/// Generate time data in different formats.
{attribute: 'hide_all_locals'}
FUNCTION_BLOCK PUBLIC DateTime
VAR
  local_system_time : Tc2_Utilities.FB_LocalSystemTime;
  get_system_time : Tc2_System.GetSystemTime;
  time_zone_info : Tc2_Utilities.FB_GetTimeZoneInformation;
  local_Time : Tc2_Utilities.FB_SystemTimeToTzSpecificLocalTime;
  local_system_time_valid : Tc2_Standard.R_Trig;
  utc_time : Tc2_Utilities.FB_TzSpecificLocalTimeToFileTime;
END_VAR

// Get local system time
local_system_time(
	sNetID  :=  '',
	bEnable :=  TRUE,
	dwCycle :=  1,
	dwOpt :=  1,
	tTimeout:= Tc2_System.Default_Ads_Timeout
);

// Get timezone information
time_zone_info(
	sNetID := '',
	bExecute := TRUE,
	tTimeout := Tc2_System.Default_Ads_Timeout
);

// Convert local time to utc time
utc_time(
	in := THIS^.AsLocalFileTime,
	tzInfo := time_zone_info.tzInfo
);
  
// Finished retrieving time data
local_system_time_valid(Clk := local_system_time.bValid);

/// Returns local time as `Tc2_Utilities.T_FILETIME`.
{attribute 'monitoring':='variable'}
PROPERTY AsLocalFileTime : Tc2_Utilities.T_FILETIME
GET
AsLocalFileTime := SYSTEMTIME_TO_FILETIME(THIS^.AsLocalSystemTime);
END_GET
END_PROPERTY

/// Returns local time as `Tc2_Utilities.TIMESTRUCT`.
{attribute 'monitoring':='variable'}
PROPERTY AsLocalSystemTime : Tc2_Utilities.TIMESTRUCT
GET
AsLocalSystemTime := local_system_time.systemTime;
END_GET
END_PROPERTY

/// Returns local time as string.
{attribute 'monitoring':='variable'}
PROPERTY AsLocalSystemTimeString : Tc2_System.T_MAXSTRING
GET
AsLocalSystemTimeString := Tc2_Utilities.SYSTEMTIME_TO_STRING(THIS^.AsLocalSystemTime);
END_GET
END_PROPERTY

/// Returns UTC time as `Tc2_Utilities.T_FILETIME`.
{attribute 'monitoring':='variable'}
PROPERTY AsUtcFileTime : Tc2_Utilities.T_FILETIME
GET
AsUtcFileTime := utc_time.out;
END_GET
END_PROPERTY

/// When calling `DateTime` the first time, it takes some time until all time and timezone information is available.
/// `Done` is `TRUE` for one cycle, once all the data is ready. 
{attribute 'monitoring':='call'}
PROPERTY Done : BOOL
GET
Done := local_system_time_valid.Q;
END_GET
END_PROPERTY

// Replaces placeholders in format string by the actual time values.
{attribute 'hide_all_locals'}
{attribute 'hide'}
METHOD PRIVATE ReplaceFormatPlaceholder : STRING
VAR_INPUT
  format : STRING;
  length : INT;
  timeType : STRING(1);
END_VAR
VAR_INST
  i : INT;
  replaceString : STRING;
  timeString : STRING;
END_VAR
VAR
  localSystemTime : Tc2_Utilities.TIMESTRUCT;
END_VAR
localSystemTime := THIS^.AsLocalSystemTime;

IF    timeType = 'Y'  THEN timeString := TO_STRING(localSystemTime.wYear); 
ELSIF timeType = 'M'  THEN timeString := TO_STRING(localSystemTime.wMonth); 
ELSIF timeType = 'D'  THEN timeString := TO_STRING(localSystemTime.wDay); 
ELSIF timeType = 'h'  THEN timeString := TO_STRING(localSystemTime.wHour); 
ELSIF timeType = 'm'  THEN timeString := TO_STRING(localSystemTime.wMinute); 
ELSIF timeType = 's'  THEN timeString := TO_STRING(localSystemTime.wSecond); 
ELSIF timeType = 'i'  THEN timeString := TO_STRING(localSystemTime.wMilliseconds); 
ELSE
  timeString:='';
END_IF

replaceString := '';

IF length > Tc2_Standard.LEN(timeString) THEN
  FOR i:=1 TO length - Tc2_Standard.LEN(timeString) DO
    replaceString := Tc2_Standard.CONCAT(replaceString, '0');
  END_FOR
  replaceString := Tc2_Standard.CONCAT(replaceString, timeString);
ELSE
  replaceString := Tc2_Standard.RIGHT(timeString, length);
END_IF

ReplaceFormatPlaceholder := Tc2_Standard.REPLACE(format, replaceString, length, Tc2_Standard.FIND(format, timeType));
END_METHOD

/// Returns a formatted string containing the actual time information 
/// - `Y` : year
/// - `M` : month
/// - `D` : day
/// - `h` : hour 
/// - `m` : minute
/// - `s` : second
/// - `i` : millisecond
/// 
/// Example:    
/// _YYMMDD-hh:mm:ss:iii_   
/// => _20210812-12:30:22:123_
{attribute 'hide_all_locals'}
METHOD ToFormatString : Tc2_System.T_MaxString
VAR_INPUT
  /// Format the timestamp should have.
  format : STRING;
END_VAR
VAR_INST
  inputString : STRING;
  c : STRING(1);
  formattedString : Tc2_System.T_MaxString;
END_VAR
VAR
  year : INT := 0;
  month : INT := 0;
  day : INT := 0;
  hour : INT := 0;
  minute : INT := 0;
  second : INT := 0;
  millisecond : INT := 0;
END_VAR
VAR CONSTANT
  ValidFormat : STRING := 'YMDhms';
END_VAR
// Parses "format" and returns a adequatly formatted string containing the time information
inputString := format;

WHILE Tc2_Standard.LEN(inputString) > 0 DO
  c := Tc2_Standard.LEFT(inputString, 1);
  
  IF    c = 'Y' THEN year := year + 1;
  ELSIF c = 'M' THEN month := month + 1;
  ELSIF c = 'D' THEN day := day + 1;
  ELSIF c = 'h' THEN hour := hour + 1;
  ELSIF c = 'm' THEN minute := minute + 1;
  ELSIF c = 's' THEN second := second + 1;
  ELSIF c = 'i' THEN millisecond := millisecond + 1;
  END_IF
  
  inputString := Tc2_Standard.DELETE(inputString, 1, 1);
END_WHILE

formattedString := ReplaceFormatPlaceholder(format, year, 'Y');
formattedString := ReplaceFormatPlaceholder(formattedString, month, 'M');
formattedString := ReplaceFormatPlaceholder(formattedString, day, 'D');
formattedString := ReplaceFormatPlaceholder(formattedString, hour, 'h');
formattedString := ReplaceFormatPlaceholder(formattedString, minute, 'm');
formattedString := ReplaceFormatPlaceholder(formattedString, second, 's');
formattedString := ReplaceFormatPlaceholder(formattedString, millisecond, 'i');

ToFormatString := formattedString;
END_METHOD

END_FUNCTION_BLOCK

(* stored: Version 1.1.0.1
   POU DateTime: Id {a1415746-5629-4121-889a-c1e5c1a14e0f}, SpecialFunc None
   Property AsLocalFileTime: Id {b720c5a4-1100-428c-a7e2-41b868a071ff}
   Get Get: Id {b1a2f50c-6988-4b92-b085-85a9004a1612}
   Property AsLocalSystemTime: Id {b4e1e9aa-2a1f-48d2-b550-fd1086ff3fdd}
   Get Get: Id {fa4393c2-6109-4d9e-b2fa-3ad7b62ed2f8}
   Property AsLocalSystemTimeString: Id {5369c665-8e43-47f8-90ac-6a20e91f9b15}
   Get Get: Id {35077403-8c65-49e5-bc6c-f3059db8d48d}
   Property AsUtcFileTime: Id {5d7980f5-7958-42bc-8ff9-2ff8df224d75}
   Get Get: Id {8be667d4-bf9f-48c4-8ca8-698f7b715d73}
   Property Done: Id {8f1defae-bf58-4f56-90d2-4c21f4d99c0d}
   Get Get: Id {af33a3a4-b3f8-4a12-a02f-9f9071d422ae}
   Method ReplaceFormatPlaceholder: Id {0cd85094-5af1-4c37-9111-0c2d17463a35}
   Method ToFormatString: Id {8e5c5f29-5e99-4676-80b8-ceef73719a56} *)
